(* PLC project  *)

CONFIGURATION Application
  RESOURCE Application ON PLC
    TASK EtherCAT_Task(INTERVAL := T#4ms, PRIORITY := 1);
    PROGRAM Main WITH EtherCAT_Task : Main;
  END_RESOURCE
END_CONFIGURATION
